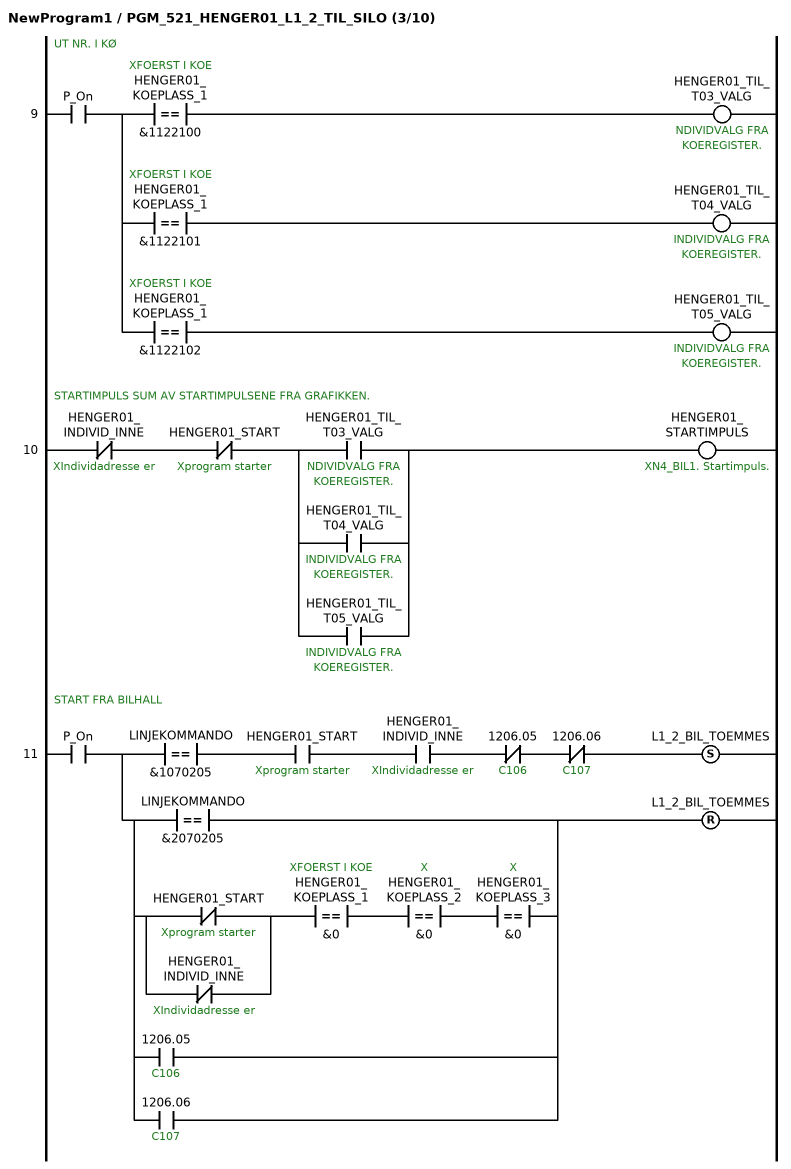
; [picture p600: NewProgram1 / PGM_521_HENGER01_L1_2_TIL_SILO, rungs 9-11]
; rung 9: UT NR. I KØ
LD P_On
OUT TR0
AND=L(301) HENGER01_KOEPLASS_1 &1122100  ; XFOERST I KOE
OUT HENGER01_TIL_T03_VALG  ; NDIVIDVALG FRA KOEREGISTER.
LD TR0
AND=L(301) HENGER01_KOEPLASS_1 &1122101  ; XFOERST I KOE
OUT HENGER01_TIL_T04_VALG  ; INDIVIDVALG FRA KOEREGISTER.
LD TR0
AND=L(301) HENGER01_KOEPLASS_1 &1122102  ; XFOERST I KOE
OUT HENGER01_TIL_T05_VALG  ; INDIVIDVALG FRA KOEREGISTER.
; rung 10: STARTIMPULS SUM AV STARTIMPULSENE FRA GRAFIKKEN.
LDNOT HENGER01_INDIVID_INNE  ; XIndividadresse er
ANDNOT HENGER01_START  ; Xprogram starter
LD HENGER01_TIL_T03_VALG  ; NDIVIDVALG FRA KOEREGISTER.
OR HENGER01_TIL_T04_VALG  ; INDIVIDVALG FRA KOEREGISTER.
OR HENGER01_TIL_T05_VALG  ; INDIVIDVALG FRA KOEREGISTER.
ANDLD
OUT HENGER01_STARTIMPULS  ; XN4_BIL1. Startimpuls.
; rung 11: START FRA BILHALL
LD P_On
OUT TR0
AND=L(301) LINJEKOMMANDO &1070205
AND HENGER01_START  ; Xprogram starter
AND HENGER01_INDIVID_INNE  ; XIndividadresse er
ANDNOT 1206.05  ; C106
ANDNOT 1206.06  ; C107
SET L1_2_BIL_TOEMMES
LD TR0
LD=L(301) LINJEKOMMANDO &2070205
LDNOT HENGER01_START  ; Xprogram starter
ORNOT HENGER01_INDIVID_INNE  ; XIndividadresse er
AND=(300) HENGER01_KOEPLASS_1 &0  ; XFOERST I KOE
AND=(300) HENGER01_KOEPLASS_2 &0  ; X
AND=(300) HENGER01_KOEPLASS_3 &0  ; X
ORLD
OR 1206.05  ; C106
OR 1206.06  ; C107
ANDLD
RSET L1_2_BIL_TOEMMES

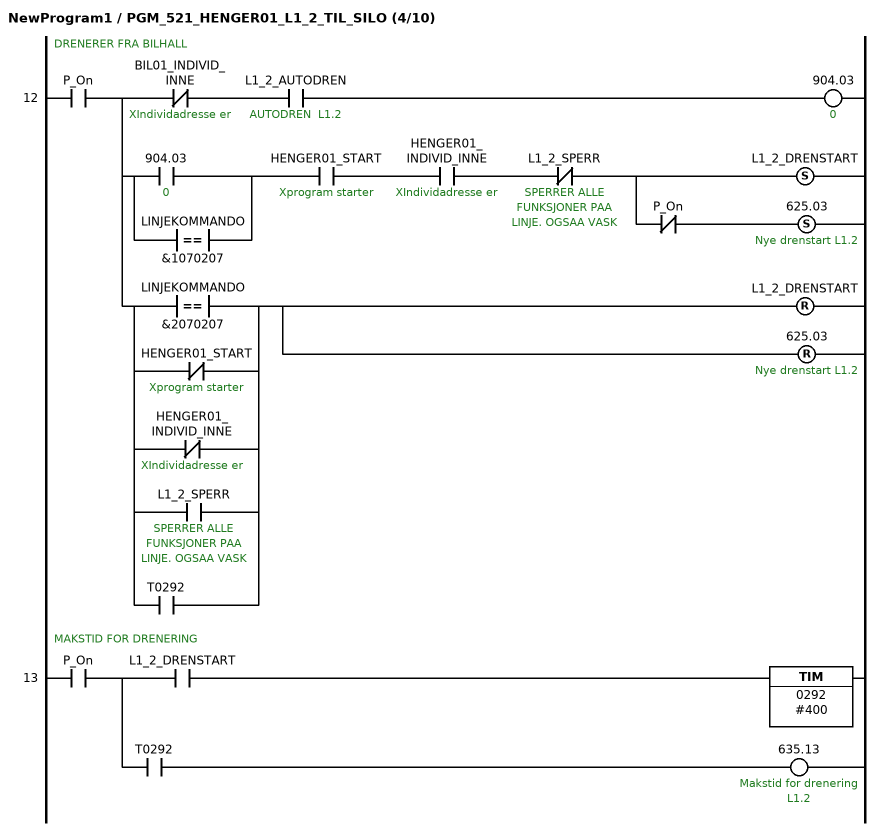
; rung 12: DRENERER FRA BILHALL
LD P_On
OUT TR0
ANDNOT BIL01_INDIVID_INNE  ; XIndividadresse er
AND L1_2_AUTODREN  ; AUTODREN  L1.2
OUT 904.03  ; 0
LD TR0
LD 904.03  ; 0
OR=L(301) LINJEKOMMANDO &1070207
ANDLD
AND HENGER01_START  ; Xprogram starter
AND HENGER01_INDIVID_INNE  ; XIndividadresse er
ANDNOT L1_2_SPERR  ; SPERRER ALLE FUNKSJONER PAA LINJE. OGSAA VASK
SET L1_2_DRENSTART
ANDNOT P_On
SET 625.03  ; Nye drenstart L1.2
LD TR0
LD=L(301) LINJEKOMMANDO &2070207
ORNOT HENGER01_START  ; Xprogram starter
ORNOT HENGER01_INDIVID_INNE  ; XIndividadresse er
OR L1_2_SPERR  ; SPERRER ALLE FUNKSJONER PAA LINJE. OGSAA VASK
OR T0292
ANDLD
RSET L1_2_DRENSTART
RSET 625.03  ; Nye drenstart L1.2
; rung 13: MAKSTID FOR DRENERING
LD P_On
OUT TR0
AND L1_2_DRENSTART
TIM 0292 #400
LD TR0
AND T0292
OUT 635.13  ; Makstid for drenering L1.2

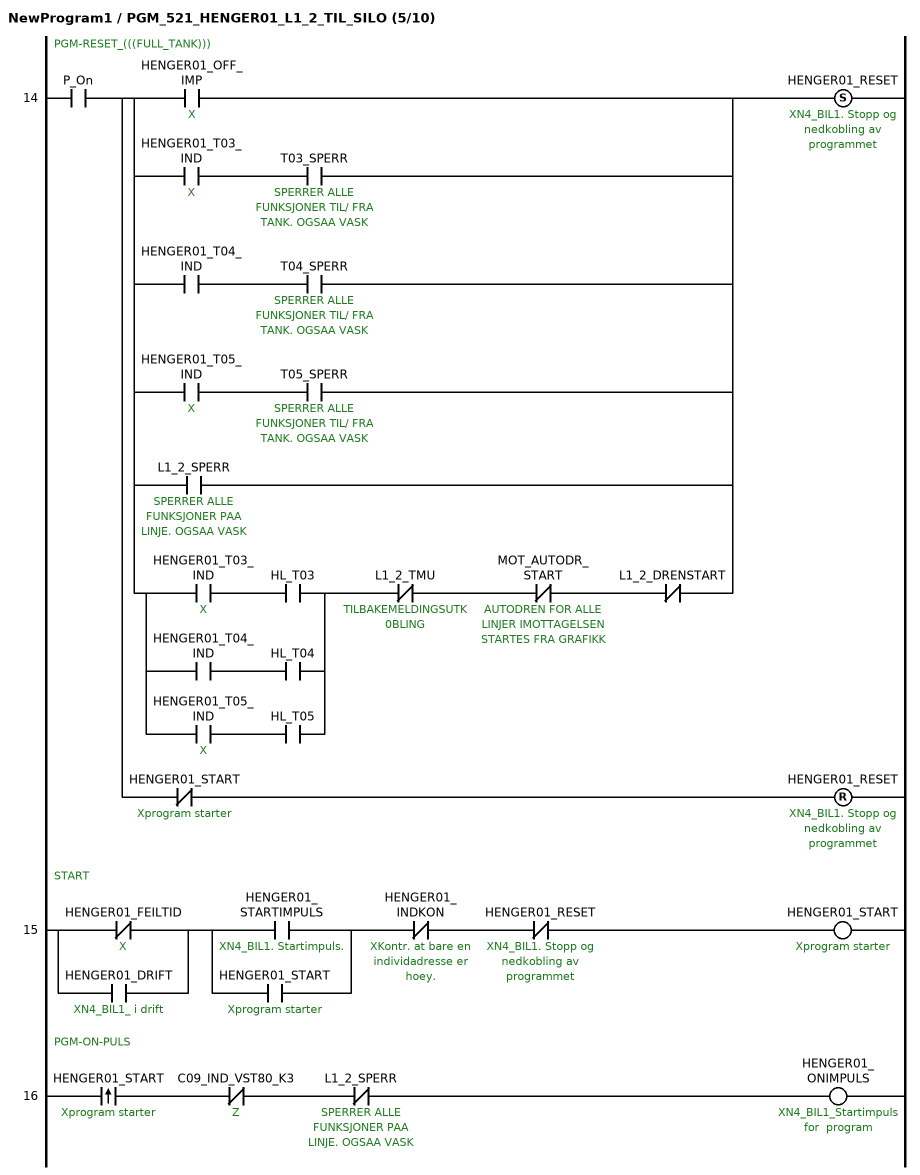
; rung 14: PGM-RESET_(((FULL_TANK)))
LD P_On
OUT TR0
LD HENGER01_OFF_IMP  ; X
LD HENGER01_T03_IND  ; X
AND T03_SPERR  ; SPERRER ALLE FUNKSJONER TIL/ FRA TANK. OGSAA VASK
ORLD
LD HENGER01_T04_IND
AND T04_SPERR  ; SPERRER ALLE FUNKSJONER TIL/ FRA TANK. OGSAA VASK
ORLD
LD HENGER01_T05_IND  ; X
AND T05_SPERR  ; SPERRER ALLE FUNKSJONER TIL/ FRA TANK. OGSAA VASK
ORLD
OR L1_2_SPERR  ; SPERRER ALLE FUNKSJONER PAA LINJE. OGSAA VASK
LD HENGER01_T03_IND  ; X
AND HL_T03
LD HENGER01_T04_IND
AND HL_T04
ORLD
LD HENGER01_T05_IND  ; X
AND HL_T05
ORLD
ANDNOT L1_2_TMU  ; TILBAKEMELDINGSUTK0BLING
ANDNOT MOT_AUTODR_START  ; AUTODREN FOR ALLE LINJER IMOTTAGELSEN STARTES FRA GRAFIKK
ANDNOT L1_2_DRENSTART
ORLD
ANDLD
SET HENGER01_RESET  ; XN4_BIL1. Stopp og nedkobling av programmet
LD TR0
ANDNOT HENGER01_START  ; Xprogram starter
RSET HENGER01_RESET  ; XN4_BIL1. Stopp og nedkobling av programmet
; rung 15: START
LDNOT HENGER01_FEILTID  ; X
OR HENGER01_DRIFT  ; XN4_BIL1_ i drift
LD HENGER01_STARTIMPULS  ; XN4_BIL1. Startimpuls.
OR HENGER01_START  ; Xprogram starter
ANDLD
ANDNOT HENGER01_INDKON  ; XKontr. at bare en individadresse er hoey.
ANDNOT HENGER01_RESET  ; XN4_BIL1. Stopp og nedkobling av programmet
OUT HENGER01_START  ; Xprogram starter
; rung 16: PGM-ON-PULS
@LD HENGER01_START  ; Xprogram starter
ANDNOT C09_IND_VST80_K3  ; Z
ANDNOT L1_2_SPERR  ; SPERRER ALLE FUNKSJONER PAA LINJE. OGSAA VASK
OUT HENGER01_ONIMPULS  ; XN4_BIL1_Startimpuls for  program

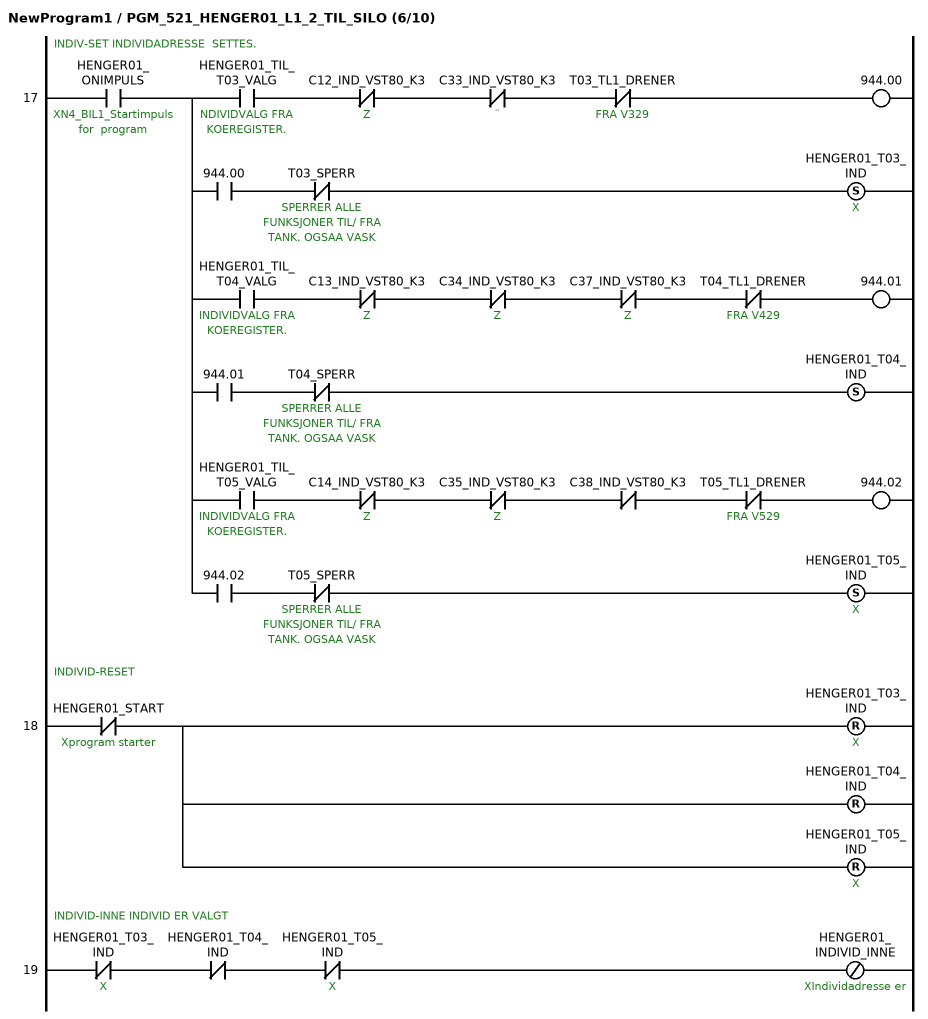
; rung 17: INDIV-SET INDIVIDADRESSE  SETTES.
LD HENGER01_ONIMPULS  ; XN4_BIL1_Startimpuls for  program
OUT TR0
AND HENGER01_TIL_T03_VALG  ; NDIVIDVALG FRA KOEREGISTER.
ANDNOT C12_IND_VST80_K3  ; Z
ANDNOT C33_IND_VST80_K3  ; ¨
ANDNOT T03_TL1_DRENER  ; FRA V329
OUT 944.00
LD TR0
AND 944.00
ANDNOT T03_SPERR  ; SPERRER ALLE FUNKSJONER TIL/ FRA TANK. OGSAA VASK
SET HENGER01_T03_IND  ; X
LD TR0
AND HENGER01_TIL_T04_VALG  ; INDIVIDVALG FRA KOEREGISTER.
ANDNOT C13_IND_VST80_K3  ; Z
ANDNOT C34_IND_VST80_K3  ; Z
ANDNOT C37_IND_VST80_K3  ; Z
ANDNOT T04_TL1_DRENER  ; FRA V429
OUT 944.01
LD TR0
AND 944.01
ANDNOT T04_SPERR  ; SPERRER ALLE FUNKSJONER TIL/ FRA TANK. OGSAA VASK
SET HENGER01_T04_IND
LD TR0
AND HENGER01_TIL_T05_VALG  ; INDIVIDVALG FRA KOEREGISTER.
ANDNOT C14_IND_VST80_K3  ; Z
ANDNOT C35_IND_VST80_K3  ; Z
ANDNOT C38_IND_VST80_K3
ANDNOT T05_TL1_DRENER  ; FRA V529
OUT 944.02
LD TR0
AND 944.02
ANDNOT T05_SPERR  ; SPERRER ALLE FUNKSJONER TIL/ FRA TANK. OGSAA VASK
SET HENGER01_T05_IND  ; X
; rung 18: INDIVID-RESET
LDNOT HENGER01_START  ; Xprogram starter
RSET HENGER01_T03_IND  ; X
RSET HENGER01_T04_IND
RSET HENGER01_T05_IND  ; X
; rung 19: INDIVID-INNE INDIVID ER VALGT
LDNOT HENGER01_T03_IND  ; X
ANDNOT HENGER01_T04_IND
ANDNOT HENGER01_T05_IND  ; X
OUTNOT HENGER01_INDIVID_INNE  ; XIndividadresse er

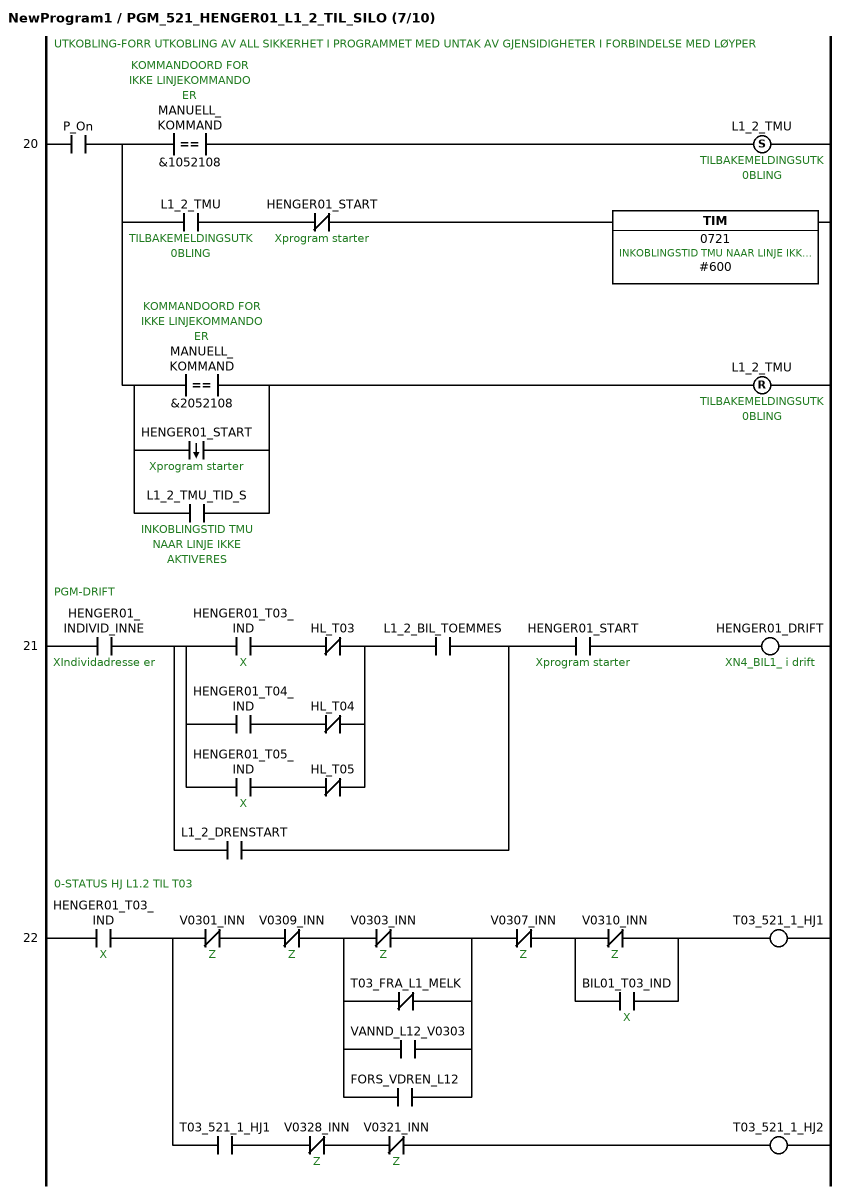
; rung 20: UTKOBLING-FORR UTKOBLING AV ALL SIKKERHET I PROGRAMMET MED UNTAK AV GJENSIDIGHETER I FORBINDELSE MED LØYPER
LD P_On
OUT TR0
AND=L(301) MANUELL_KOMMAND &1052108  ; KOMMANDOORD FOR IKKE LINJEKOMMANDOER
SET L1_2_TMU  ; TILBAKEMELDINGSUTK0BLING
LD TR0
AND L1_2_TMU  ; TILBAKEMELDINGSUTK0BLING
ANDNOT HENGER01_START  ; Xprogram starter
TIM 0721 #600  ; INKOBLINGSTID TMU NAAR LINJE IKKE AKTIVERES
LD TR0
LD=L(301) MANUELL_KOMMAND &2052108  ; KOMMANDOORD FOR IKKE LINJEKOMMANDOER
%OR HENGER01_START  ; Xprogram starter
OR L1_2_TMU_TID_S  ; INKOBLINGSTID TMU NAAR LINJE IKKE AKTIVERES
ANDLD
RSET L1_2_TMU  ; TILBAKEMELDINGSUTK0BLING
; rung 21: PGM-DRIFT
LD HENGER01_INDIVID_INNE  ; XIndividadresse er
LD HENGER01_T03_IND  ; X
ANDNOT HL_T03
LD HENGER01_T04_IND
ANDNOT HL_T04
ORLD
LD HENGER01_T05_IND  ; X
ANDNOT HL_T05
ORLD
AND L1_2_BIL_TOEMMES
OR L1_2_DRENSTART
ANDLD
AND HENGER01_START  ; Xprogram starter
OUT HENGER01_DRIFT  ; XN4_BIL1_ i drift
; rung 22: 0-STATUS HJ L1.2 TIL T03
LD HENGER01_T03_IND  ; X
OUT TR0
ANDNOT V0301_INN  ; Z
ANDNOT V0309_INN  ; Z
LDNOT V0303_INN  ; Z
ORNOT T03_FRA_L1_MELK
OR VANND_L12_V0303
OR FORS_VDREN_L12
ANDLD
ANDNOT V0307_INN  ; Z
LDNOT V0310_INN  ; Z
OR BIL01_T03_IND  ; X
ANDLD
OUT T03_521_1_HJ1
LD TR0
AND T03_521_1_HJ1
ANDNOT V0328_INN  ; Z
ANDNOT V0321_INN  ; Z
OUT T03_521_1_HJ2

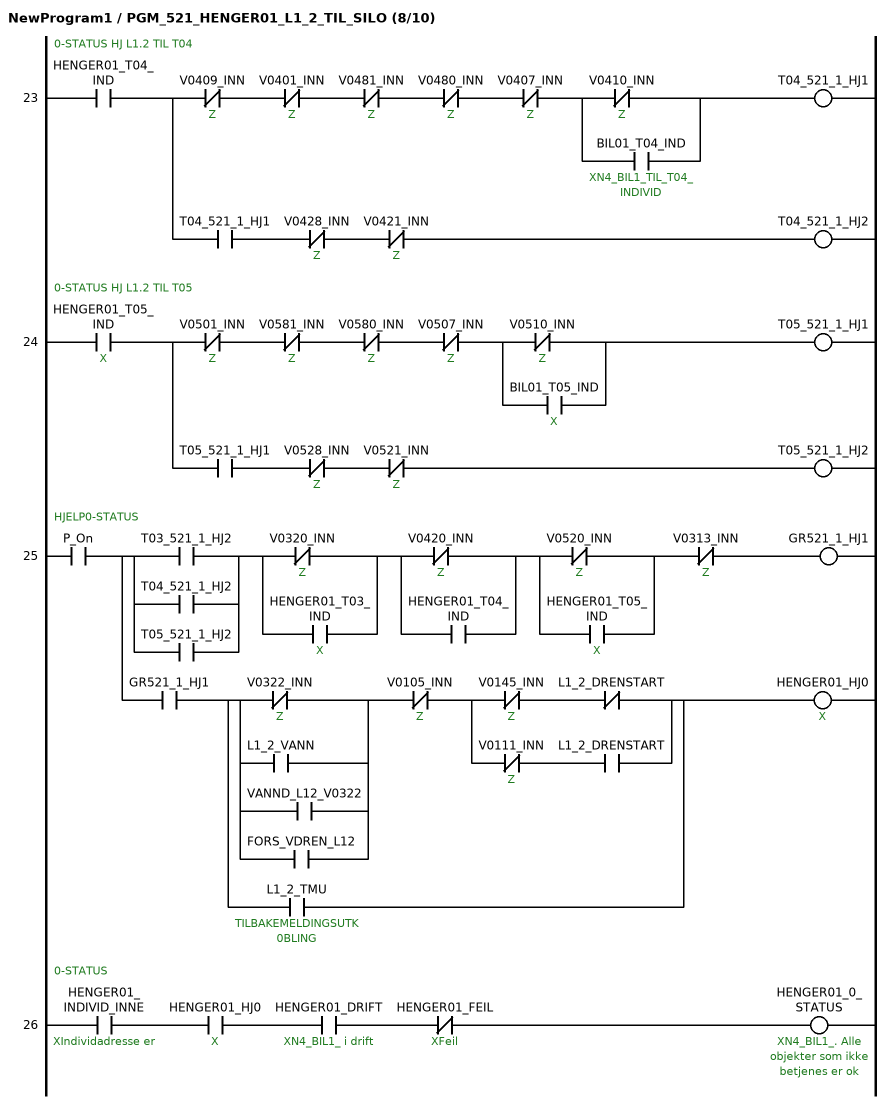
; rung 23: 0-STATUS HJ L1.2 TIL T04
LD HENGER01_T04_IND
OUT TR0
ANDNOT V0409_INN  ; Z
ANDNOT V0401_INN  ; Z
ANDNOT V0481_INN  ; Z
ANDNOT V0480_INN  ; Z
ANDNOT V0407_INN  ; Z
LDNOT V0410_INN  ; Z
OR BIL01_T04_IND  ; XN4_BIL1_TIL_T04_INDIVID
ANDLD
OUT T04_521_1_HJ1
LD TR0
AND T04_521_1_HJ1
ANDNOT V0428_INN  ; Z
ANDNOT V0421_INN  ; Z
OUT T04_521_1_HJ2
; rung 24: 0-STATUS HJ L1.2 TIL T05
LD HENGER01_T05_IND  ; X
OUT TR0
ANDNOT V0501_INN  ; Z
ANDNOT V0581_INN  ; Z
ANDNOT V0580_INN  ; Z
ANDNOT V0507_INN  ; Z
LDNOT V0510_INN  ; Z
OR BIL01_T05_IND  ; X
ANDLD
OUT T05_521_1_HJ1
LD TR0
AND T05_521_1_HJ1
ANDNOT V0528_INN  ; Z
ANDNOT V0521_INN  ; Z
OUT T05_521_1_HJ2
; rung 25: HJELP0-STATUS
LD P_On
OUT TR0
LD T03_521_1_HJ2
OR T04_521_1_HJ2
OR T05_521_1_HJ2
ANDLD
LDNOT V0320_INN  ; Z
OR HENGER01_T03_IND  ; X
ANDLD
LDNOT V0420_INN  ; Z
OR HENGER01_T04_IND
ANDLD
LDNOT V0520_INN  ; Z
OR HENGER01_T05_IND  ; X
ANDLD
ANDNOT V0313_INN  ; Z
OUT GR521_1_HJ1
LD TR0
AND GR521_1_HJ1
LDNOT V0322_INN  ; Z
OR L1_2_VANN
OR VANND_L12_V0322
OR FORS_VDREN_L12
ANDNOT V0105_INN  ; Z
LDNOT V0145_INN  ; Z
ANDNOT L1_2_DRENSTART
LDNOT V0111_INN  ; Z
AND L1_2_DRENSTART
ORLD
ANDLD
OR L1_2_TMU  ; TILBAKEMELDINGSUTK0BLING
ANDLD
OUT HENGER01_HJ0  ; X
; rung 26: 0-STATUS
LD HENGER01_INDIVID_INNE  ; XIndividadresse er
AND HENGER01_HJ0  ; X
AND HENGER01_DRIFT  ; XN4_BIL1_ i drift
ANDNOT HENGER01_FEIL  ; XFeil
OUT HENGER01_0_STATUS  ; XN4_BIL1_. Alle objekter som ikke betjenes er ok

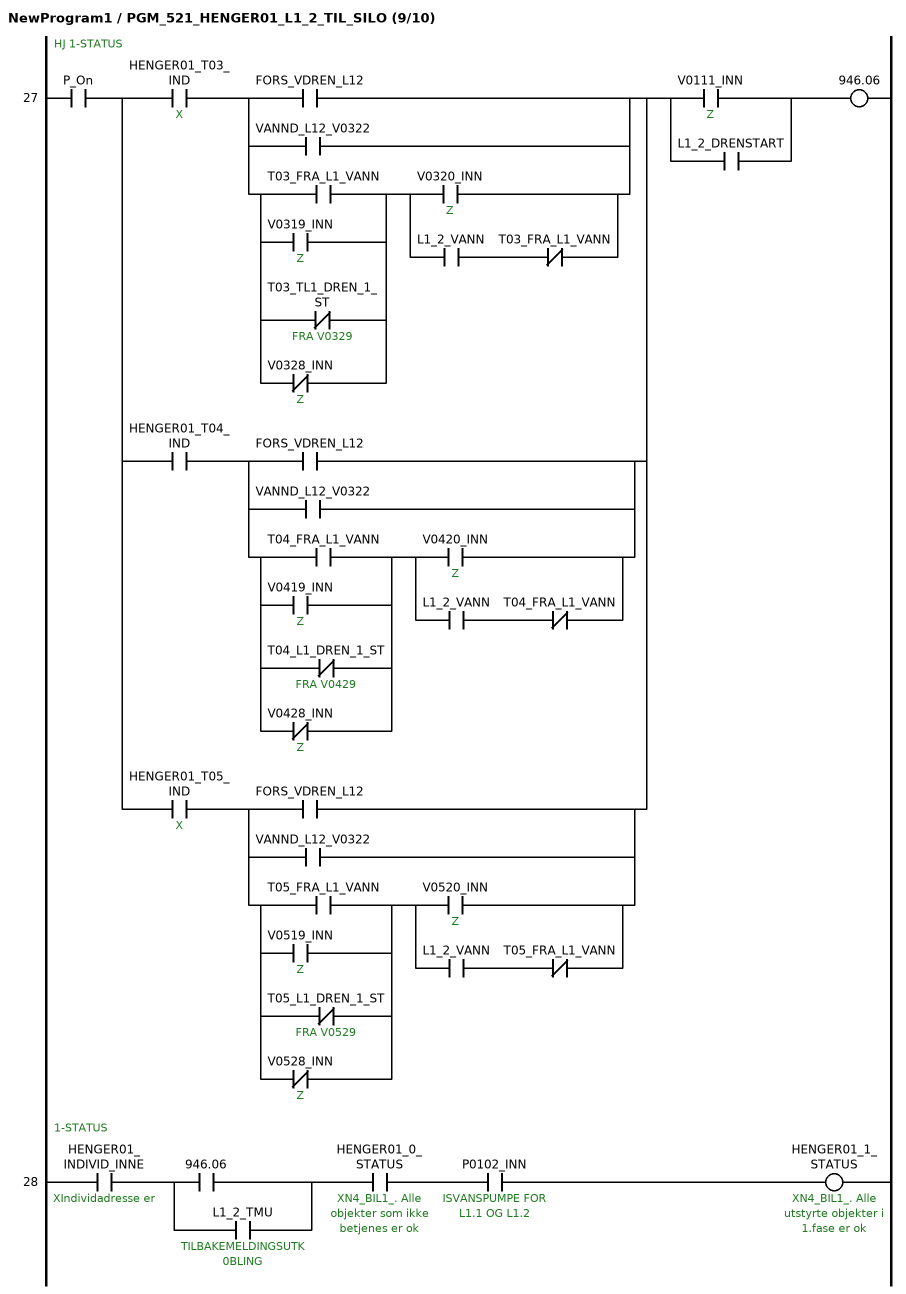
; rung 27: HJ 1-STATUS
LD P_On
LD HENGER01_T03_IND  ; X
LD FORS_VDREN_L12
OR VANND_L12_V0322
LD T03_FRA_L1_VANN
OR V0319_INN  ; Z
ORNOT T03_TL1_DREN_1_ST  ; FRA V0329
ORNOT V0328_INN  ; Z
LD V0320_INN  ; Z
LD L1_2_VANN
ANDNOT T03_FRA_L1_VANN
ORLD
ANDLD
ORLD
ANDLD
LD HENGER01_T04_IND
LD FORS_VDREN_L12
OR VANND_L12_V0322
LD T04_FRA_L1_VANN
OR V0419_INN  ; Z
ORNOT T04_L1_DREN_1_ST  ; FRA V0429
ORNOT V0428_INN  ; Z
LD V0420_INN  ; Z
LD L1_2_VANN
ANDNOT T04_FRA_L1_VANN
ORLD
ANDLD
ORLD
ANDLD
ORLD
LD HENGER01_T05_IND  ; X
LD FORS_VDREN_L12
OR VANND_L12_V0322
LD T05_FRA_L1_VANN
OR V0519_INN  ; Z
ORNOT T05_L1_DREN_1_ST  ; FRA V0529
ORNOT V0528_INN  ; Z
LD V0520_INN  ; Z
LD L1_2_VANN
ANDNOT T05_FRA_L1_VANN
ORLD
ANDLD
ORLD
ANDLD
ORLD
ANDLD
LD V0111_INN  ; Z
OR L1_2_DRENSTART
ANDLD
OUT 946.06
; rung 28: 1-STATUS
LD HENGER01_INDIVID_INNE  ; XIndividadresse er
LD 946.06
OR L1_2_TMU  ; TILBAKEMELDINGSUTK0BLING
ANDLD
AND HENGER01_0_STATUS  ; XN4_BIL1_. Alle objekter som ikke betjenes er ok
AND P0102_INN  ; ISVANSPUMPE FOR L1.1 OG L1.2
OUT HENGER01_1_STATUS  ; XN4_BIL1_. Alle utstyrte objekter i 1.fase er ok

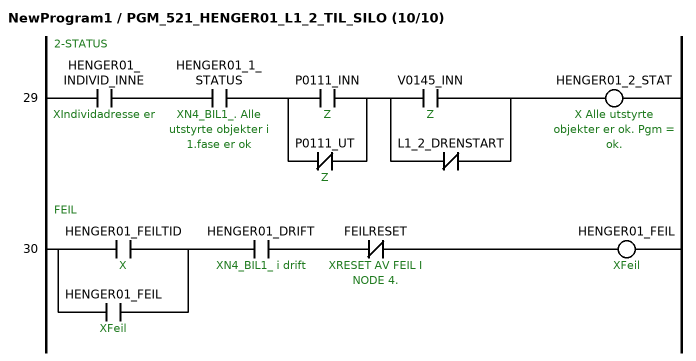
; rung 29: 2-STATUS
LD HENGER01_INDIVID_INNE  ; XIndividadresse er
AND HENGER01_1_STATUS  ; XN4_BIL1_. Alle utstyrte objekter i 1.fase er ok
LD P0111_INN  ; Z
ORNOT P0111_UT  ; Z
ANDLD
LD V0145_INN  ; Z
ORNOT L1_2_DRENSTART
ANDLD
OUT HENGER01_2_STAT  ; X Alle utstyrte objekter er ok. Pgm = ok.
; rung 30: FEIL
LD HENGER01_FEILTID  ; X
OR HENGER01_FEIL  ; XFeil
AND HENGER01_DRIFT  ; XN4_BIL1_ i drift
ANDNOT FEILRESET  ; XRESET AV FEIL I NODE 4.
OUT HENGER01_FEIL  ; XFeil

### Section V0114_P0111

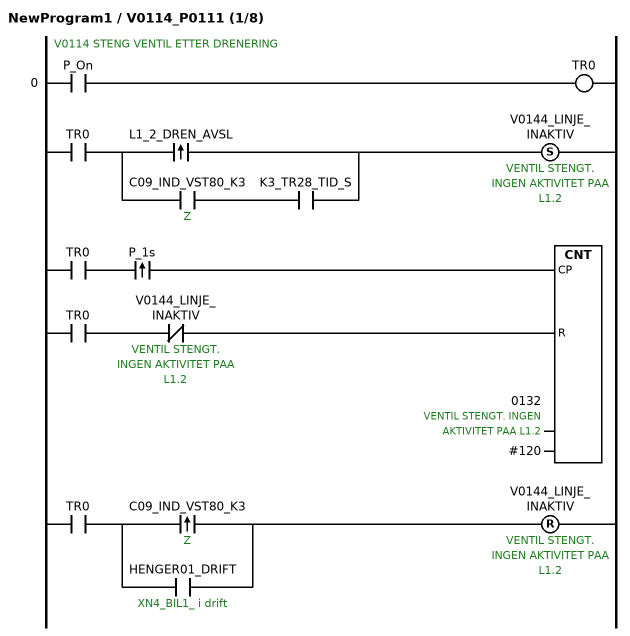
; rung 0: V0114 STENG VENTIL ETTER DRENERING
LD P_On
OUT TR0
@LD L1_2_DREN_AVSL
LD C09_IND_VST80_K3  ; Z
AND K3_TR28_TID_S
ORLD
ANDLD
SET V0144_LINJE_INAKTIV  ; VENTIL STENGT. INGEN AKTIVITET PAA L1.2
LD TR0
@AND P_1s
LD TR0
ANDNOT V0144_LINJE_INAKTIV  ; VENTIL STENGT. INGEN AKTIVITET PAA L1.2
CNT 0132 #120  ; VENTIL STENGT. INGEN AKTIVITET PAA L1.2
LD TR0
@LD C09_IND_VST80_K3  ; Z
OR HENGER01_DRIFT  ; XN4_BIL1_ i drift
ANDLD
RSET V0144_LINJE_INAKTIV  ; VENTIL STENGT. INGEN AKTIVITET PAA L1.2

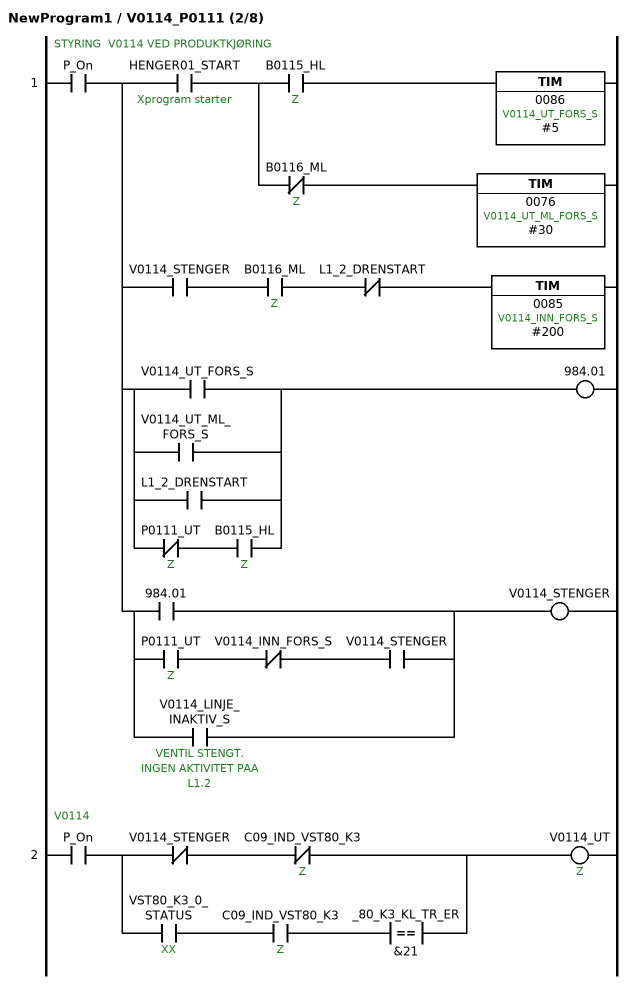
; rung 1: STYRING  V0114 VED PRODUKTKJØRING
LD P_On
OUT TR0
AND HENGER01_START  ; Xprogram starter
OUT TR1
AND B0115_HL  ; Z
TIM 0086 #5  ; V0114_UT_FORS_S
LD TR1
ANDNOT B0116_ML  ; Z
TIM 0076 #30  ; V0114_UT_ML_FORS_S
LD TR0
AND V0114_STENGER
AND B0116_ML  ; Z
ANDNOT L1_2_DRENSTART
TIM 0085 #200  ; V0114_INN_FORS_S
LD TR0
LD V0114_UT_FORS_S
OR V0114_UT_ML_FORS_S
OR L1_2_DRENSTART
LDNOT P0111_UT  ; Z
AND B0115_HL  ; Z
ORLD
ANDLD
OUT 984.01
LD TR0
LD 984.01
LD P0111_UT  ; Z
ANDNOT V0114_INN_FORS_S
AND V0114_STENGER
ORLD
OR V0114_LINJE_INAKTIV_S  ; VENTIL STENGT. INGEN AKTIVITET PAA L1.2
ANDLD
OUT V0114_STENGER
; rung 2: V0114
LD P_On
LDNOT V0114_STENGER
ANDNOT C09_IND_VST80_K3  ; Z
LD VST80_K3_0_STATUS  ; XX
AND C09_IND_VST80_K3  ; Z
AND=(300) _80_K3_KL_TR_ER &21
ORLD
ANDLD
OUT V0114_UT  ; Z

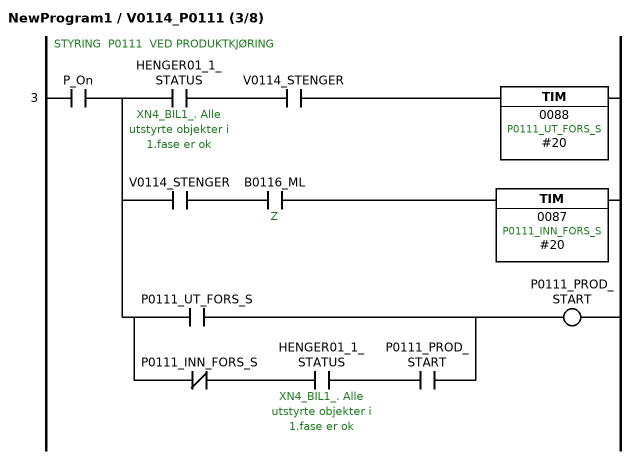
; rung 3: STYRING  P0111  VED PRODUKTKJØRING
LD P_On
OUT TR0
AND HENGER01_1_STATUS  ; XN4_BIL1_. Alle utstyrte objekter i 1.fase er ok
AND V0114_STENGER
TIM 0088 #20  ; P0111_UT_FORS_S
LD TR0
AND V0114_STENGER
AND B0116_ML  ; Z
TIM 0087 #20  ; P0111_INN_FORS_S
LD TR0
LD P0111_UT_FORS_S
LDNOT P0111_INN_FORS_S
AND HENGER01_1_STATUS  ; XN4_BIL1_. Alle utstyrte objekter i 1.fase er ok
AND P0111_PROD_START
ORLD
ANDLD
OUT P0111_PROD_START

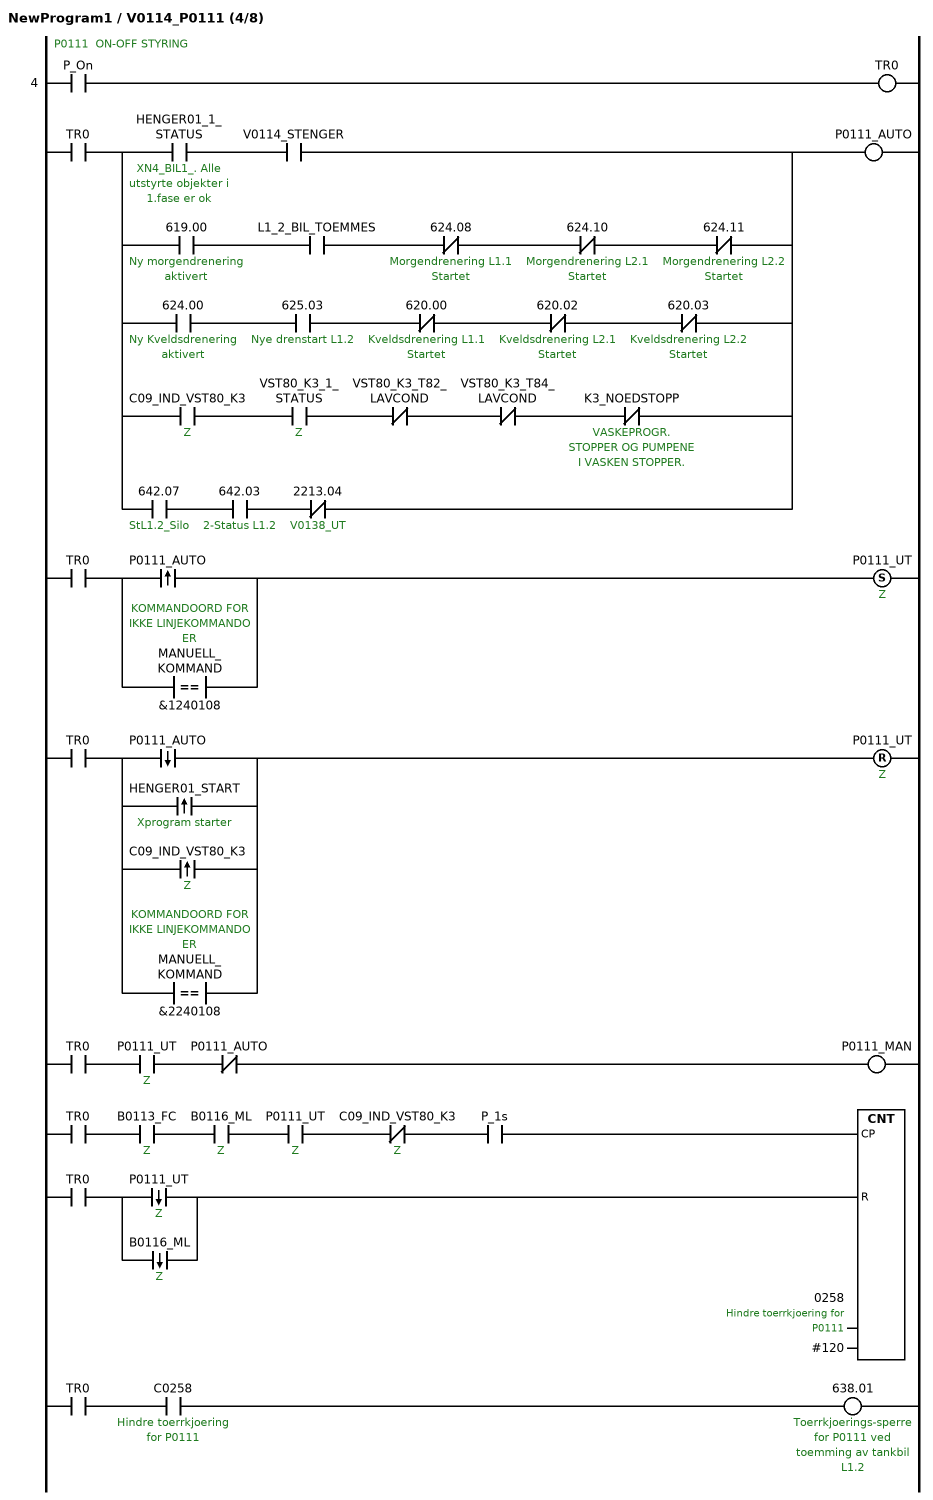
; rung 4: P0111  ON-OFF STYRING
LD P_On
OUT TR0
LD HENGER01_1_STATUS  ; XN4_BIL1_. Alle utstyrte objekter i 1.fase er ok
AND V0114_STENGER
LD 619.00  ; Ny morgendrenering aktivert
AND L1_2_BIL_TOEMMES
ANDNOT 624.08  ; Morgendrenering L1.1 Startet
ANDNOT 624.10  ; Morgendrenering L2.1 Startet
ANDNOT 624.11  ; Morgendrenering L2.2 Startet
ORLD
LD 624.00  ; Ny Kveldsdrenering aktivert
AND 625.03  ; Nye drenstart L1.2
ANDNOT 620.00  ; Kveldsdrenering L1.1 Startet
ANDNOT 620.02  ; Kveldsdrenering L2.1 Startet
ANDNOT 620.03  ; Kveldsdrenering L2.2 Startet
ORLD
LD C09_IND_VST80_K3  ; Z
AND VST80_K3_1_STATUS  ; Z
ANDNOT VST80_K3_T82_LAVCOND
ANDNOT VST80_K3_T84_LAVCOND
ANDNOT K3_NOEDSTOPP  ; VASKEPROGR. STOPPER OG PUMPENE I VASKEN STOPPER.
ORLD
LD 642.07  ; StL1.2_Silo
AND 642.03  ; 2-Status L1.2
ANDNOT 2213.04  ; V0138_UT
ORLD
ANDLD
OUT P0111_AUTO
LD TR0
@LD P0111_AUTO
OR=L(301) MANUELL_KOMMAND &1240108  ; KOMMANDOORD FOR IKKE LINJEKOMMANDOER
ANDLD
SET P0111_UT  ; Z
LD TR0
%LD P0111_AUTO
@OR HENGER01_START  ; Xprogram starter
@OR C09_IND_VST80_K3  ; Z
OR=L(301) MANUELL_KOMMAND &2240108  ; KOMMANDOORD FOR IKKE LINJEKOMMANDOER
ANDLD
RSET P0111_UT  ; Z
LD TR0
AND P0111_UT  ; Z
ANDNOT P0111_AUTO
OUT P0111_MAN
LD TR0
AND B0113_FC  ; Z
AND B0116_ML  ; Z
AND P0111_UT  ; Z
ANDNOT C09_IND_VST80_K3  ; Z
AND P_1s
LD TR0
%LD P0111_UT  ; Z
%OR B0116_ML  ; Z
ANDLD
CNT 0258 #120  ; Hindre toerrkjoering for P0111
LD TR0
AND C0258  ; Hindre toerrkjoering for P0111
OUT 638.01  ; Toerrkjoerings-sperre for P0111 ved toemming av tankbil L1.2

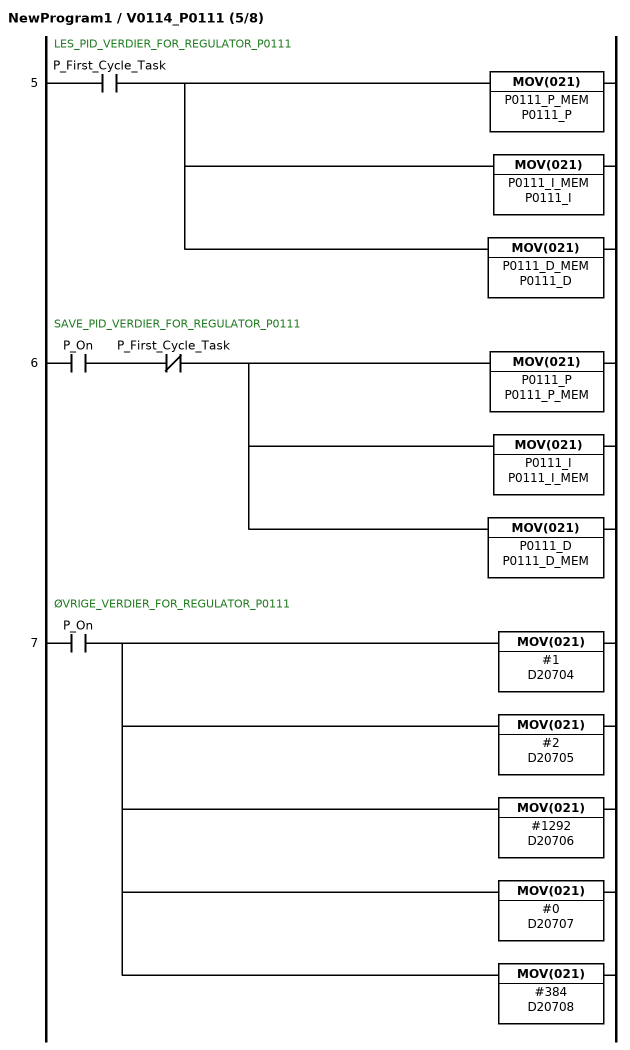
; rung 5: LES_PID_VERDIER_FOR_REGULATOR_P0111
LD P_First_Cycle_Task
MOV(021) P0111_P_MEM P0111_P
MOV(021) P0111_I_MEM P0111_I
MOV(021) P0111_D_MEM P0111_D
; rung 6: SAVE_PID_VERDIER_FOR_REGULATOR_P0111
LD P_On
ANDNOT P_First_Cycle_Task
MOV(021) P0111_P P0111_P_MEM
MOV(021) P0111_I P0111_I_MEM
MOV(021) P0111_D P0111_D_MEM
; rung 7: ØVRIGE_VERDIER_FOR_REGULATOR_P0111
LD P_On
MOV(021) #1 D20704
MOV(021) #2 D20705
MOV(021) #1292 D20706
MOV(021) #0 D20707
MOV(021) #384 D20708

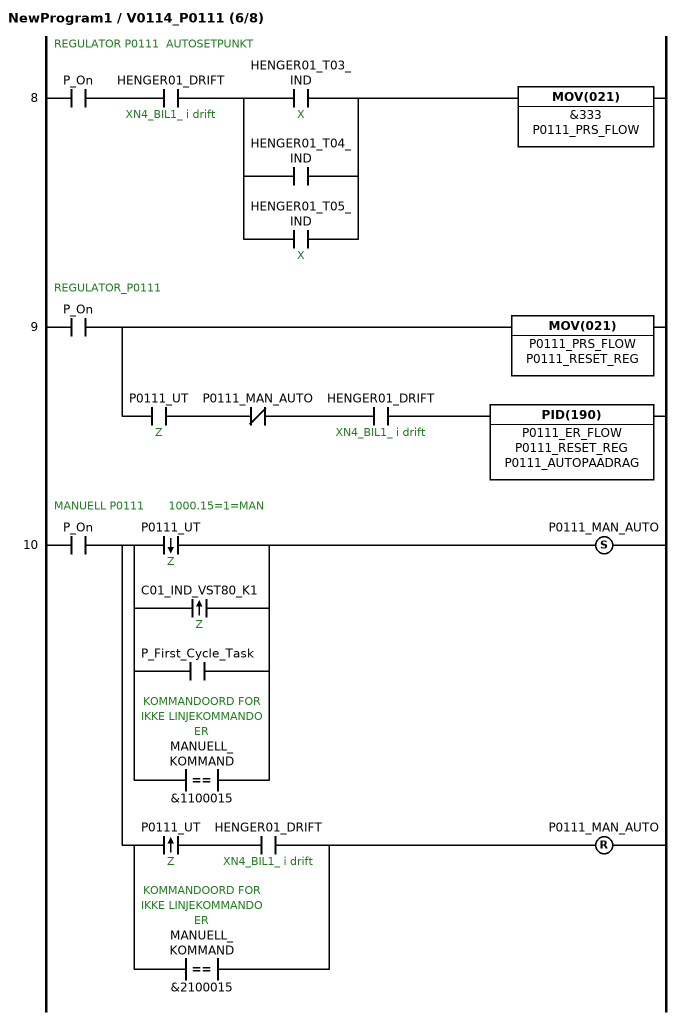
; rung 8: REGULATOR P0111  AUTOSETPUNKT
LD P_On
AND HENGER01_DRIFT  ; XN4_BIL1_ i drift
LD HENGER01_T03_IND  ; X
OR HENGER01_T04_IND
OR HENGER01_T05_IND  ; X
ANDLD
MOV(021) &333 P0111_PRS_FLOW
; rung 9: REGULATOR_P0111
LD P_On
MOV(021) P0111_PRS_FLOW P0111_RESET_REG
AND P0111_UT  ; Z
ANDNOT P0111_MAN_AUTO
AND HENGER01_DRIFT  ; XN4_BIL1_ i drift
PID(190) P0111_ER_FLOW P0111_RESET_REG P0111_AUTOPAADRAG
; rung 10: MANUELL P0111       1000.15=1=MAN
LD P_On
OUT TR0
%LD P0111_UT  ; Z
@OR C01_IND_VST80_K1  ; Z
OR P_First_Cycle_Task
OR=L(301) MANUELL_KOMMAND &1100015  ; KOMMANDOORD FOR IKKE LINJEKOMMANDOER
ANDLD
SET P0111_MAN_AUTO
LD TR0
@LD P0111_UT  ; Z
AND HENGER01_DRIFT  ; XN4_BIL1_ i drift
OR=L(301) MANUELL_KOMMAND &2100015  ; KOMMANDOORD FOR IKKE LINJEKOMMANDOER
ANDLD
RSET P0111_MAN_AUTO

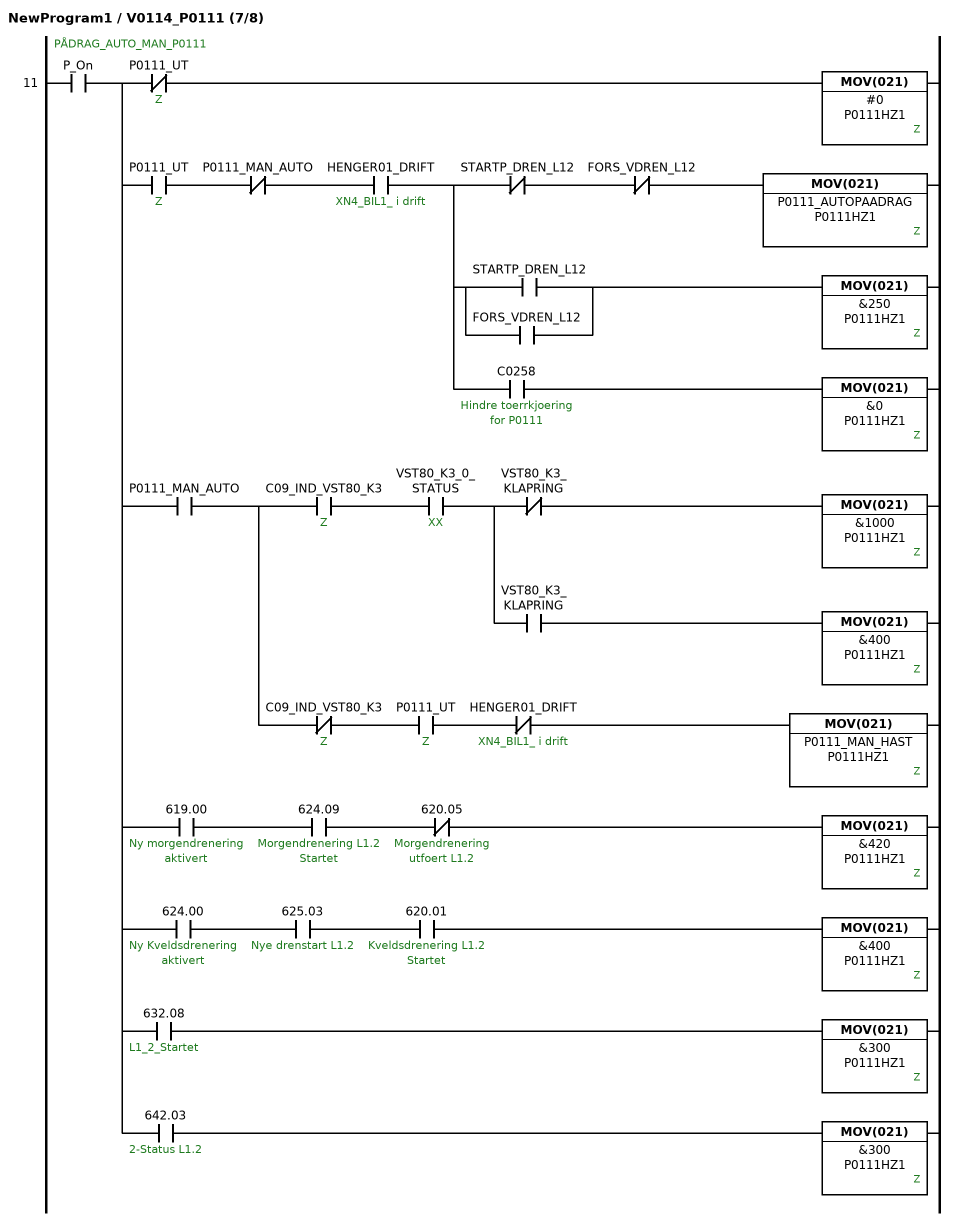
; rung 11: PÅDRAG_AUTO_MAN_P0111
LD P_On
OUT TR0
ANDNOT P0111_UT  ; Z
MOV(021) #0 P0111HZ1  ; Z
LD TR0
AND P0111_UT  ; Z
ANDNOT P0111_MAN_AUTO
AND HENGER01_DRIFT  ; XN4_BIL1_ i drift
OUT TR1
ANDNOT STARTP_DREN_L12
ANDNOT FORS_VDREN_L12
MOV(021) P0111_AUTOPAADRAG P0111HZ1  ; Z
LD TR1
LD STARTP_DREN_L12
OR FORS_VDREN_L12
ANDLD
MOV(021) &250 P0111HZ1  ; Z
LD TR1
AND C0258  ; Hindre toerrkjoering for P0111
MOV(021) &0 P0111HZ1  ; Z
LD TR0
AND P0111_MAN_AUTO
OUT TR1
AND C09_IND_VST80_K3  ; Z
AND VST80_K3_0_STATUS  ; XX
OUT TR2
ANDNOT VST80_K3_KLAPRING
MOV(021) &1000 P0111HZ1  ; Z
LD TR2
AND VST80_K3_KLAPRING
MOV(021) &400 P0111HZ1  ; Z
LD TR1
ANDNOT C09_IND_VST80_K3  ; Z
AND P0111_UT  ; Z
ANDNOT HENGER01_DRIFT  ; XN4_BIL1_ i drift
MOV(021) P0111_MAN_HAST P0111HZ1  ; Z
LD TR0
AND 619.00  ; Ny morgendrenering aktivert
AND 624.09  ; Morgendrenering L1.2 Startet
ANDNOT 620.05  ; Morgendrenering utfoert L1.2
MOV(021) &420 P0111HZ1  ; Z
LD TR0
AND 624.00  ; Ny Kveldsdrenering aktivert
AND 625.03  ; Nye drenstart L1.2
AND 620.01  ; Kveldsdrenering L1.2 Startet
MOV(021) &400 P0111HZ1  ; Z
LD TR0
AND 632.08  ; L1_2_Startet
MOV(021) &300 P0111HZ1  ; Z
LD TR0
AND 642.03  ; 2-Status L1.2
MOV(021) &300 P0111HZ1  ; Z

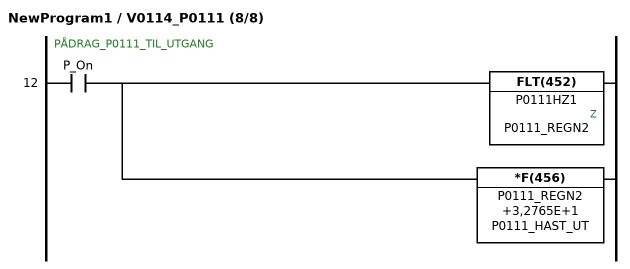
; rung 12: PÅDRAG_P0111_TIL_UTGANG
LD P_On
FLT(452) P0111HZ1 P0111_REGN2  ; Z
*F(456) P0111_REGN2 +3,2765E+1 P0111_HAST_UT

### Section V151_V0154_ISV

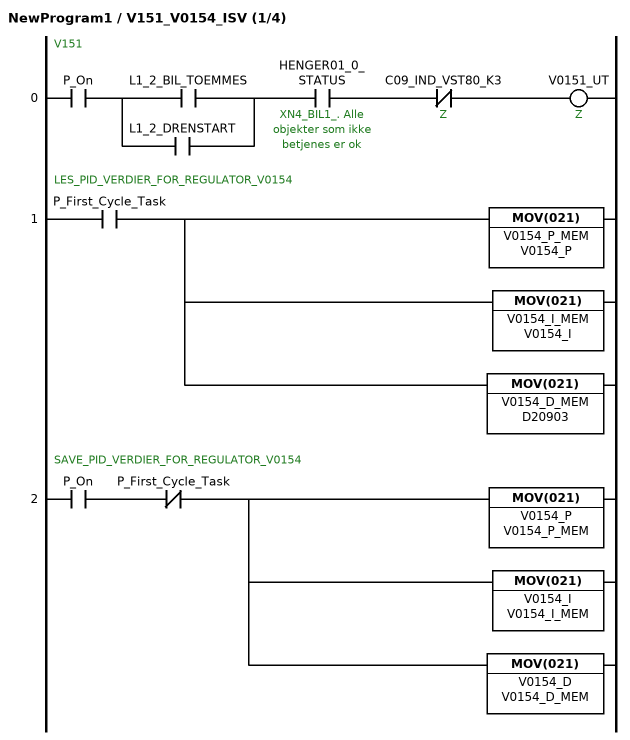
; rung 0: V151
LD P_On
LD L1_2_BIL_TOEMMES
OR L1_2_DRENSTART
ANDLD
AND HENGER01_0_STATUS  ; XN4_BIL1_. Alle objekter som ikke betjenes er ok
ANDNOT C09_IND_VST80_K3  ; Z
OUT V0151_UT  ; Z
; rung 1: LES_PID_VERDIER_FOR_REGULATOR_V0154
LD P_First_Cycle_Task
MOV(021) V0154_P_MEM V0154_P
MOV(021) V0154_I_MEM V0154_I
MOV(021) V0154_D_MEM D20903
; rung 2: SAVE_PID_VERDIER_FOR_REGULATOR_V0154
LD P_On
ANDNOT P_First_Cycle_Task
MOV(021) V0154_P V0154_P_MEM
MOV(021) V0154_I V0154_I_MEM
MOV(021) V0154_D V0154_D_MEM

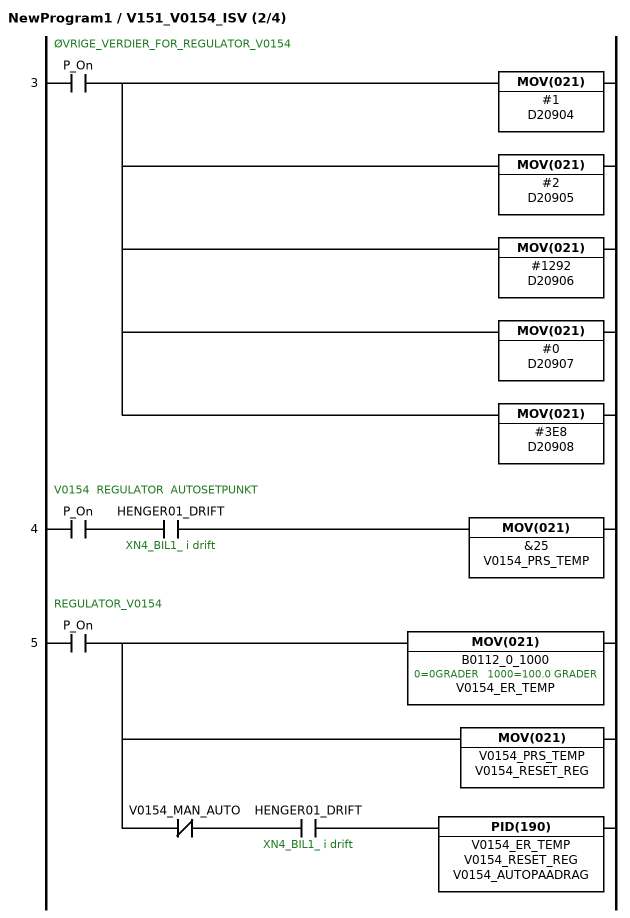
; rung 3: ØVRIGE_VERDIER_FOR_REGULATOR_V0154
LD P_On
MOV(021) #1 D20904
MOV(021) #2 D20905
MOV(021) #1292 D20906
MOV(021) #0 D20907
MOV(021) #3E8 D20908
; rung 4: V0154  REGULATOR  AUTOSETPUNKT
LD P_On
AND HENGER01_DRIFT  ; XN4_BIL1_ i drift
MOV(021) &25 V0154_PRS_TEMP
; rung 5: REGULATOR_V0154
LD P_On
MOV(021) B0112_0_1000 V0154_ER_TEMP  ; 0=0GRADER   1000=100.0 GRADER
MOV(021) V0154_PRS_TEMP V0154_RESET_REG
ANDNOT V0154_MAN_AUTO
AND HENGER01_DRIFT  ; XN4_BIL1_ i drift
PID(190) V0154_ER_TEMP V0154_RESET_REG V0154_AUTOPAADRAG

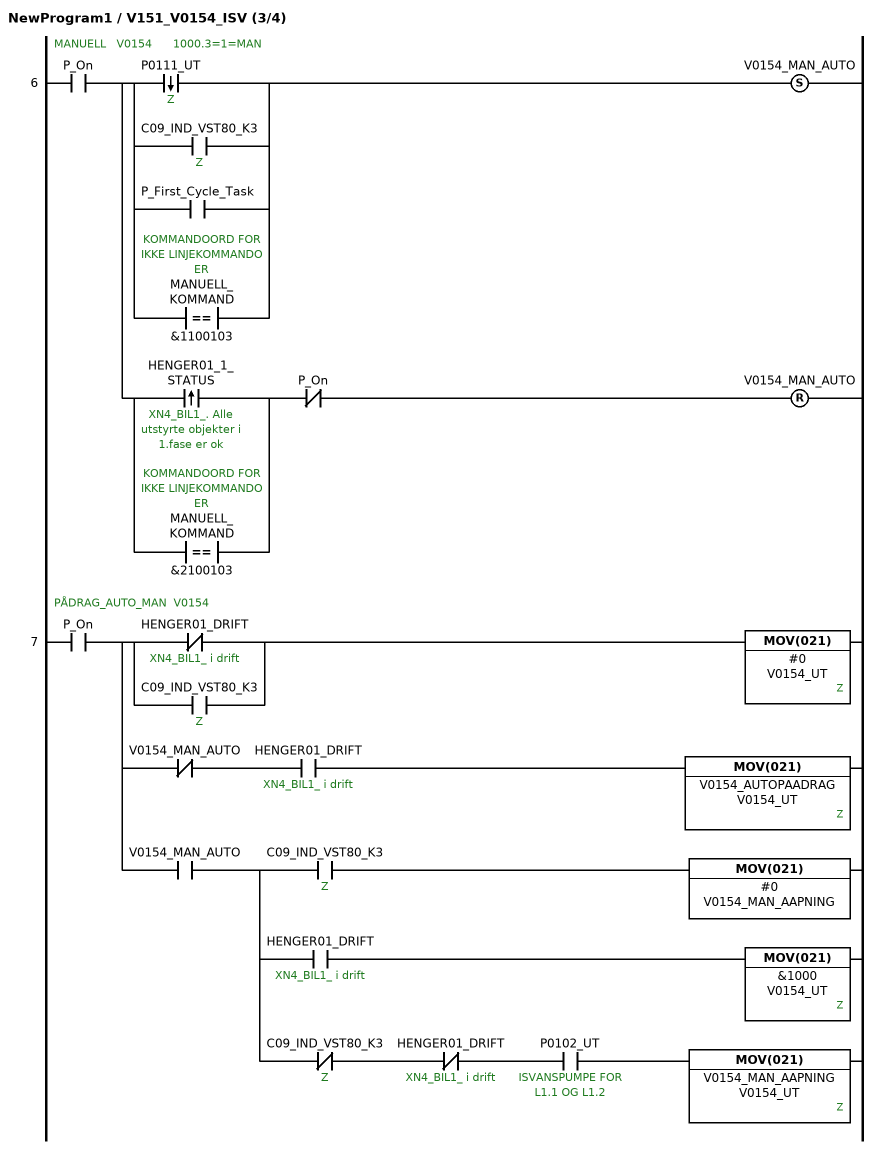
; rung 6: MANUELL   V0154      1000.3=1=MAN
LD P_On
OUT TR0
%LD P0111_UT  ; Z
OR C09_IND_VST80_K3  ; Z
OR P_First_Cycle_Task
OR=L(301) MANUELL_KOMMAND &1100103  ; KOMMANDOORD FOR IKKE LINJEKOMMANDOER
ANDLD
SET V0154_MAN_AUTO
LD TR0
@LD HENGER01_1_STATUS  ; XN4_BIL1_. Alle utstyrte objekter i 1.fase er ok
OR=L(301) MANUELL_KOMMAND &2100103  ; KOMMANDOORD FOR IKKE LINJEKOMMANDOER
ANDLD
ANDNOT P_On
RSET V0154_MAN_AUTO
; rung 7: PÅDRAG_AUTO_MAN  V0154
LD P_On
OUT TR0
LDNOT HENGER01_DRIFT  ; XN4_BIL1_ i drift
OR C09_IND_VST80_K3  ; Z
ANDLD
MOV(021) #0 V0154_UT  ; Z
LD TR0
ANDNOT V0154_MAN_AUTO
AND HENGER01_DRIFT  ; XN4_BIL1_ i drift
MOV(021) V0154_AUTOPAADRAG V0154_UT  ; Z
LD TR0
AND V0154_MAN_AUTO
OUT TR0
AND C09_IND_VST80_K3  ; Z
MOV(021) #0 V0154_MAN_AAPNING
LD TR0
AND HENGER01_DRIFT  ; XN4_BIL1_ i drift
MOV(021) &1000 V0154_UT  ; Z
LD TR0
ANDNOT C09_IND_VST80_K3  ; Z
ANDNOT HENGER01_DRIFT  ; XN4_BIL1_ i drift
AND P0102_UT  ; ISVANSPUMPE FOR L1.1 OG L1.2
MOV(021) V0154_MAN_AAPNING V0154_UT  ; Z

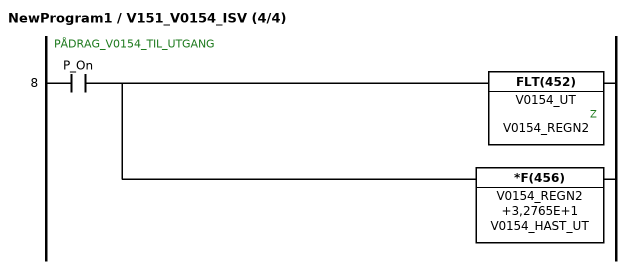
; rung 8: PÅDRAG_V0154_TIL_UTGANG
LD P_On
FLT(452) V0154_UT V0154_REGN2  ; Z
*F(456) V0154_REGN2 +3,2765E+1 V0154_HAST_UT

### Section PGM_522_BIL02_TIL_SILO

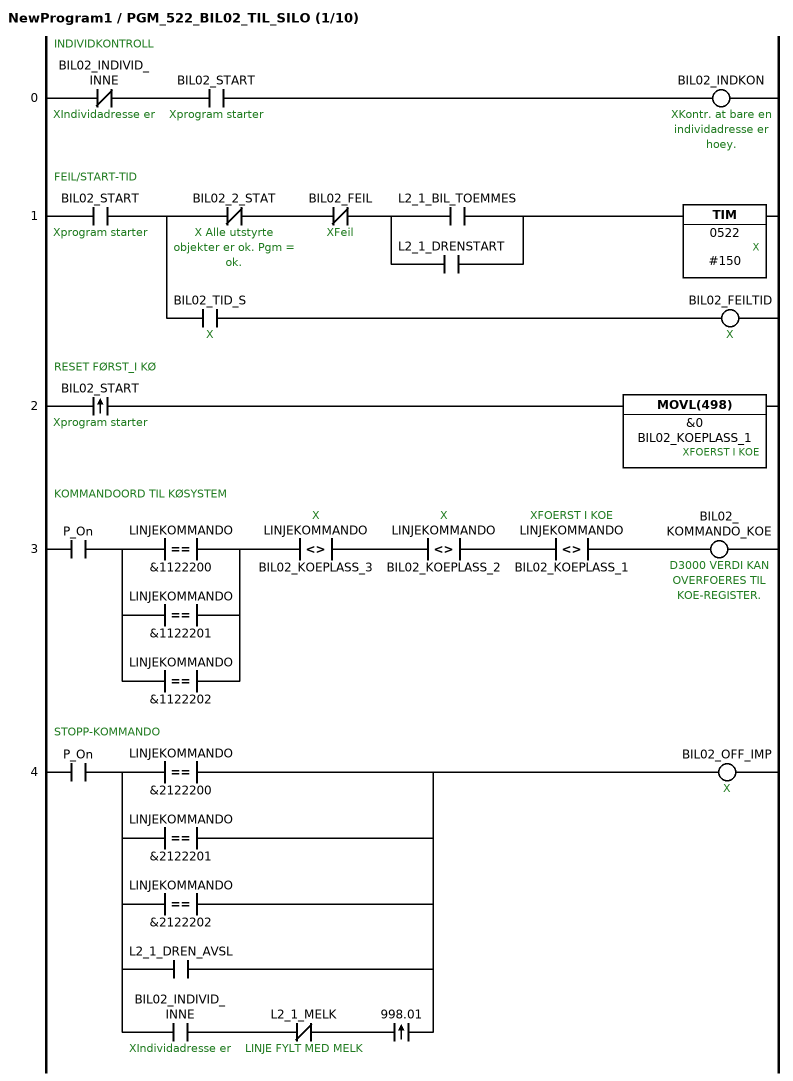
; rung 0: INDIVIDKONTROLL
LDNOT BIL02_INDIVID_INNE  ; XIndividadresse er
AND BIL02_START  ; Xprogram starter
OUT BIL02_INDKON  ; XKontr. at bare en individadresse er hoey.
; rung 1: FEIL/START-TID
LD BIL02_START  ; Xprogram starter
OUT TR0
ANDNOT BIL02_2_STAT  ; X Alle utstyrte objekter er ok. Pgm = ok.
ANDNOT BIL02_FEIL  ; XFeil
LD L2_1_BIL_TOEMMES
OR L2_1_DRENSTART
ANDLD
TIM 0522 #150  ; X
LD TR0
AND BIL02_TID_S  ; X
OUT BIL02_FEILTID  ; X
; rung 2: RESET FØRST_I KØ
@LD BIL02_START  ; Xprogram starter
MOVL(498) &0 BIL02_KOEPLASS_1  ; XFOERST I KOE
; rung 3: KOMMANDOORD TIL KØSYSTEM
LD P_On
LD=L(301) LINJEKOMMANDO &1122200
OR=L(301) LINJEKOMMANDO &1122201
OR=L(301) LINJEKOMMANDO &1122202
ANDLD
AND<>L(306) LINJEKOMMANDO BIL02_KOEPLASS_3  ; X
AND<>L(306) LINJEKOMMANDO BIL02_KOEPLASS_2  ; X
AND<>L(306) LINJEKOMMANDO BIL02_KOEPLASS_1  ; XFOERST I KOE
OUT BIL02_KOMMANDO_KOE  ; D3000 VERDI KAN OVERFOERES TIL KOE-REGISTER.
; rung 4: STOPP-KOMMANDO
LD P_On
LD=L(301) LINJEKOMMANDO &2122200
OR=L(301) LINJEKOMMANDO &2122201
OR=L(301) LINJEKOMMANDO &2122202
OR L2_1_DREN_AVSL
LD BIL02_INDIVID_INNE  ; XIndividadresse er
ANDNOT L2_1_MELK  ; LINJE FYLT MED MELK
@AND 998.01
ORLD
ANDLD
OUT BIL02_OFF_IMP  ; X

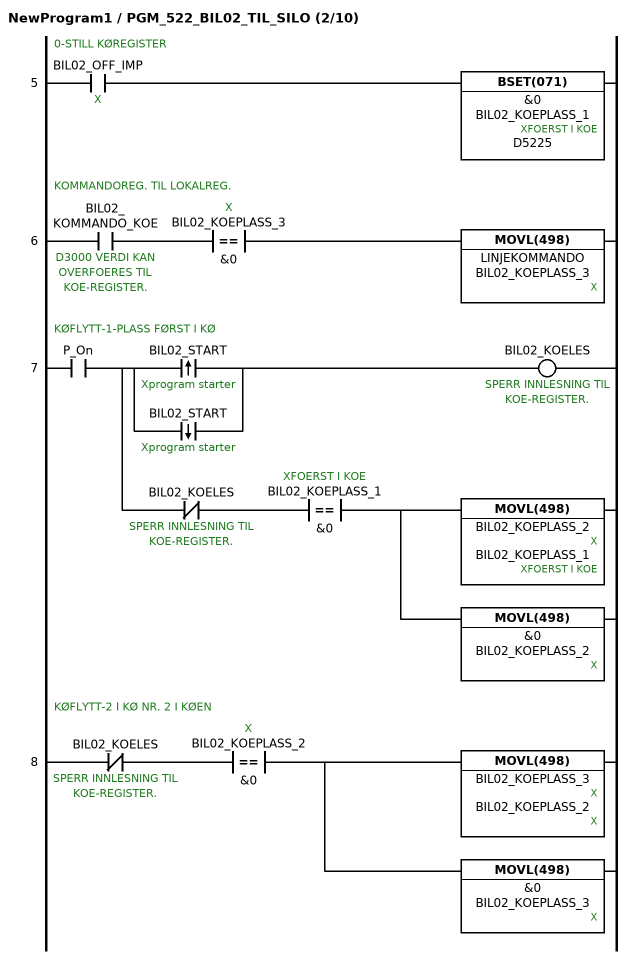
; rung 5: 0-STILL KØREGISTER
LD BIL02_OFF_IMP  ; X
BSET(071) &0 BIL02_KOEPLASS_1 D5225  ; XFOERST I KOE
; rung 6: KOMMANDOREG. TIL LOKALREG.
LD BIL02_KOMMANDO_KOE  ; D3000 VERDI KAN OVERFOERES TIL KOE-REGISTER.
AND=L(301) BIL02_KOEPLASS_3 &0  ; X
MOVL(498) LINJEKOMMANDO BIL02_KOEPLASS_3  ; X
; rung 7: KØFLYTT-1-PLASS FØRST I KØ
LD P_On
OUT TR0
@LD BIL02_START  ; Xprogram starter
%OR BIL02_START  ; Xprogram starter
ANDLD
OUT BIL02_KOELES  ; SPERR INNLESNING TIL KOE-REGISTER.
LD TR0
ANDNOT BIL02_KOELES  ; SPERR INNLESNING TIL KOE-REGISTER.
AND=L(301) BIL02_KOEPLASS_1 &0  ; XFOERST I KOE
MOVL(498) BIL02_KOEPLASS_2 BIL02_KOEPLASS_1  ; X, XFOERST I KOE
MOVL(498) &0 BIL02_KOEPLASS_2  ; X
; rung 8: KØFLYTT-2 I KØ NR. 2 I KØEN
LDNOT BIL02_KOELES  ; SPERR INNLESNING TIL KOE-REGISTER.
AND=L(301) BIL02_KOEPLASS_2 &0  ; X
MOVL(498) BIL02_KOEPLASS_3 BIL02_KOEPLASS_2  ; X
MOVL(498) &0 BIL02_KOEPLASS_3  ; X

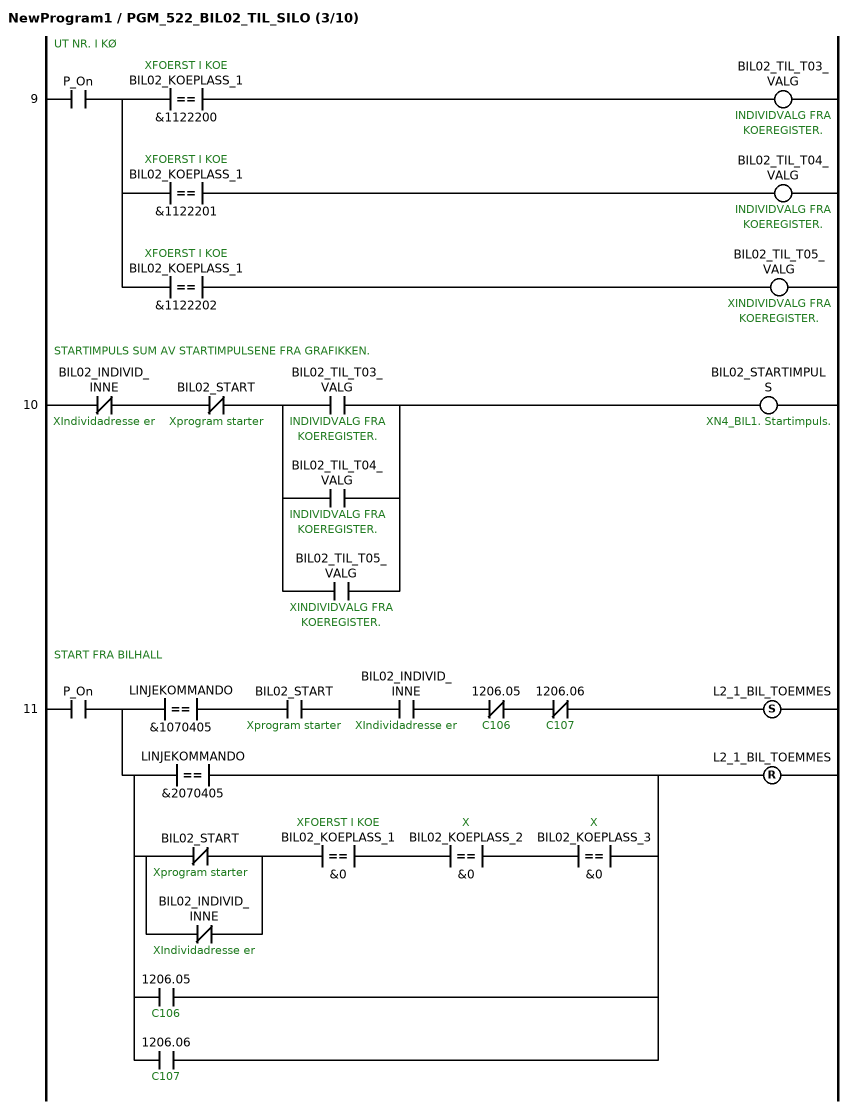
; rung 9: UT NR. I KØ
LD P_On
OUT TR0
AND=L(301) BIL02_KOEPLASS_1 &1122200  ; XFOERST I KOE
OUT BIL02_TIL_T03_VALG  ; INDIVIDVALG FRA KOEREGISTER.
LD TR0
AND=L(301) BIL02_KOEPLASS_1 &1122201  ; XFOERST I KOE
OUT BIL02_TIL_T04_VALG  ; INDIVIDVALG FRA KOEREGISTER.
LD TR0
AND=L(301) BIL02_KOEPLASS_1 &1122202  ; XFOERST I KOE
OUT BIL02_TIL_T05_VALG  ; XINDIVIDVALG FRA KOEREGISTER.
; rung 10: STARTIMPULS SUM AV STARTIMPULSENE FRA GRAFIKKEN.
LDNOT BIL02_INDIVID_INNE  ; XIndividadresse er
ANDNOT BIL02_START  ; Xprogram starter
LD BIL02_TIL_T03_VALG  ; INDIVIDVALG FRA KOEREGISTER.
OR BIL02_TIL_T04_VALG  ; INDIVIDVALG FRA KOEREGISTER.
OR BIL02_TIL_T05_VALG  ; XINDIVIDVALG FRA KOEREGISTER.
ANDLD
OUT BIL02_STARTIMPULS  ; XN4_BIL1. Startimpuls.
; rung 11: START FRA BILHALL
LD P_On
OUT TR0
AND=L(301) LINJEKOMMANDO &1070405
AND BIL02_START  ; Xprogram starter
AND BIL02_INDIVID_INNE  ; XIndividadresse er
ANDNOT 1206.05  ; C106
ANDNOT 1206.06  ; C107
SET L2_1_BIL_TOEMMES
LD TR0
LD=L(301) LINJEKOMMANDO &2070405
LDNOT BIL02_START  ; Xprogram starter
ORNOT BIL02_INDIVID_INNE  ; XIndividadresse er
AND=(300) BIL02_KOEPLASS_1 &0  ; XFOERST I KOE
AND=(300) BIL02_KOEPLASS_2 &0  ; X
AND=(300) BIL02_KOEPLASS_3 &0  ; X
ORLD
OR 1206.05  ; C106
OR 1206.06  ; C107
ANDLD
RSET L2_1_BIL_TOEMMES

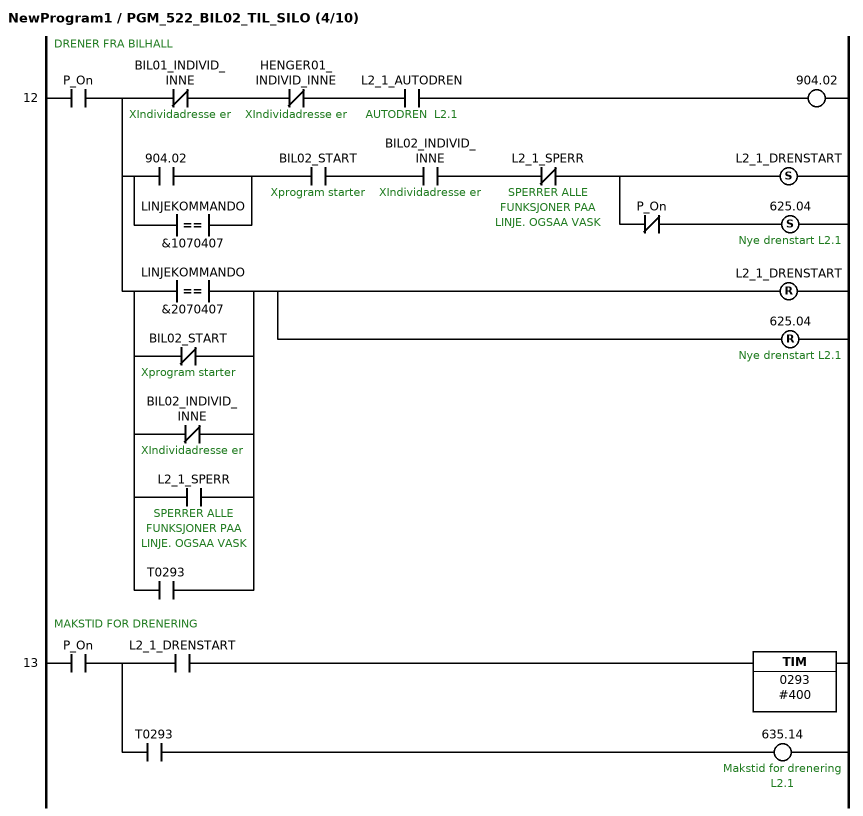
; rung 12: DRENER FRA BILHALL
LD P_On
OUT TR0
ANDNOT BIL01_INDIVID_INNE  ; XIndividadresse er
ANDNOT HENGER01_INDIVID_INNE  ; XIndividadresse er
AND L2_1_AUTODREN  ; AUTODREN  L2.1
OUT 904.02
LD TR0
LD 904.02
OR=L(301) LINJEKOMMANDO &1070407
ANDLD
AND BIL02_START  ; Xprogram starter
AND BIL02_INDIVID_INNE  ; XIndividadresse er
ANDNOT L2_1_SPERR  ; SPERRER ALLE FUNKSJONER PAA LINJE. OGSAA VASK
SET L2_1_DRENSTART
ANDNOT P_On
SET 625.04  ; Nye drenstart L2.1
LD TR0
LD=L(301) LINJEKOMMANDO &2070407
ORNOT BIL02_START  ; Xprogram starter
ORNOT BIL02_INDIVID_INNE  ; XIndividadresse er
OR L2_1_SPERR  ; SPERRER ALLE FUNKSJONER PAA LINJE. OGSAA VASK
OR T0293
ANDLD
RSET L2_1_DRENSTART
RSET 625.04  ; Nye drenstart L2.1
; rung 13: MAKSTID FOR DRENERING
LD P_On
OUT TR0
AND L2_1_DRENSTART
TIM 0293 #400
LD TR0
AND T0293
OUT 635.14  ; Makstid for drenering L2.1

